FUNCTION_BLOCK L3_NewPartHDLR (* Basic Function Block Type *)
  (* Standard: 61499-2 *)
  (* Version 0.0, 2014-11-04, EQUEROL, UJI *)
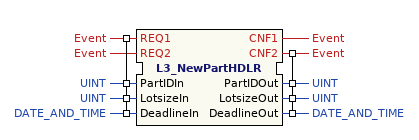
  EVENT_INPUT
    REQ1 WITH PartIDIn, LotsizeIn, DeadlineIn; (* Execution request *)
    REQ2; (* Normal Execution Request *)
  END_EVENT
  EVENT_OUTPUT
    CNF1; (* Execution confirm *)
    CNF2 WITH PartIDOut, LotsizeOut, DeadlineOut; (* Execution Confirmation *)
  END_EVENT
  VAR_INPUT
    PartIDIn : UINT; (* Identifier of the 1st part to be created *)
    LotsizeIn : UINT; (* Number of parts to be manufactured *)
    DeadlineIn : DATE_AND_TIME; (* Parts delivery deadline *)
  END_VAR
  VAR_OUTPUT
    PartIDOut : UINT; (* Part identifier *)
    LotsizeOut : UINT; (* Number of parts to be manufactured *)
    DeadlineOut : DATE_AND_TIME; (* Parts delivery date *)
  END_VAR
  VAR
    PartBuffer : ARRAY [0..9] OF UINT := [0,0,0,0,0,0,0,0,0,0]; (* Buffer to hold incoming orders's identifiers *)
    SizesBuffer : ARRAY [0..9] OF UINT := [0,0,0,0,0,0,0,0,0,0]; (* Buffer to hold incoming orders' lotsize *)
    DeadlinesBuffer : ARRAY [0..9] OF DATE_AND_TIME; (* Buffer to hold incoming orders's deadlines *)
    HeadIndex : USINT := 0; (* Index pointing to the head of the buffer *)
    TailIndex : USINT := 0; (* Index pointing to the tail of the buffer *)
    BufferSize : USINT := 10; (* Internal Variable *)
  END_VAR
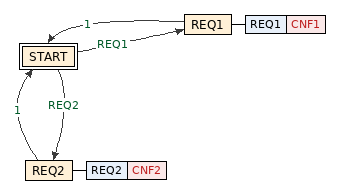
  EC_STATES
    START; (* Initial State *)
    REQ1 : REQ1 -> CNF1; (* Initialization *)
    REQ2 : REQ2 -> CNF2; (* Normal execution *)
  END_STATES
  EC_TRANSITIONS
    START TO REQ1 := REQ1;
    REQ1 TO START := 1;
    START TO REQ2 := REQ2;
    REQ2 TO START := 1;
  END_TRANSITIONS
  ALGORITHM REQ1 IN ST: (* Normally executed algorithm *)
IF PartBuffer[HeadIndex] <> PartIDIn THEN
	(*Stack the received order*)
	PartBuffer[HeadIndex] := PartIDIn;
	SizesBuffer[HeadIndex] := LotsizeIn;
	DeadlinesBuffer[HeadIndex] := DeadlineIn;

	(*PostIncrement HeadIndex*)
	HeadIndex := HeadIndex + 1;
	IF HeadIndex >= BufferSize THEN
		HeadIndex := 0;
	END_IF;

	(*Check if buffer is full*)
	IF HeadIndex = TailIndex THEN
		(*Buffer is full, HeadIndex can't be incremented*)
		IF HeadIndex = 0 THEN
			HeadIndex := BufferSize - 1;
		ELSE
			HeadIndex := HeadIndex - 1;
		END_IF;
	END_IF;
ELSE
	(*Retransmited Order, RSP event must have been lost*)
	(*Do nothing and send CNF1 event*)
END_IF;
  END_ALGORITHM
  ALGORITHM REQ2 IN ST: (* Normal execution algo *)
IF HeadIndex = TailIndex THEN
	(*Buffer is empty*)
	PartIDOut := 0;
	LotsizeOut := 0;
	DeadlineOut := DT#0-0-0-0:00:00;
ELSE
	PartIDOut := PartBuffer[TailIndex];
	LotsizeOut := SizesBuffer[TailIndex];
	DeadlineOut := DeadlinesBuffer[TailIndex];
	(*Increase tail index*)
	TailIndex := TailIndex + 1;
	IF TailIndex >= BufferSize THEN
		TailIndex := 0;
	END_IF;
END_IF;
  END_ALGORITHM
END_FUNCTION_BLOCK
